FUNCTION_BLOCK AreaOutputEx EXTENDS SectionEx
VAR_IN_OUT
	outputBuffer : ARRAY[*] OF Bundle;
END_VAR
VAR
	passConveyorPos (* AT %I* *) : REAL;
	failConveyorPos (* AT %I* *) : REAL;
	bufferConveyorPos (* AT %I* *) : REAL;
	
	step : (GET_RESULT, CHECK_RESULT, RESET);
	grade : (BYPASS, PASS, FAIL);
END_VAR
VAR
	gradeRequestString : STRING(1000);
	visionTimer : TON;
END_VAR
VAR_STAT CONSTANT
	visionTimeout : TIME := T#10S;
END_VAR

entryRefPos := bufferConveyorPos;
exitRefPos := MAX(passConveyorPos, failConveyorPos);

visionTimer(IN:= , PT:= visionTimeout, Q=> , ET=> );

SUPER^();

METHOD changeRobotsEOAT : BOOL
END_METHOD

METHOD gradeBundle : BOOL
VAR_INPUT
END_VAR
CASE grade OF
	PASS:
		//send to PASS output, LEFT
		
	BYPASS, FAIL:
		//send to FAIL output for manual correction, RIGHT
		
END_CASE
END_METHOD

METHOD initHardware : BOOL
conveyors := ADR(Hardware.allConveyors);
END_METHOD

METHOD PROTECTED load : BOOL
VAR_INPUT
	pair : REFERENCE TO PositionMaterials;
END_VAR
(*
loading takes place while the section is NOT active
materials are loaded for the next incoming bundle, not the current bundle - may differ for each section
*)
END_METHOD

METHOD PROTECTED process : BOOL
VAR
	gradingTcpData : TcpData;
END_VAR
VAR
	visionJson : STRING(1000);
	visionData : VisionFrame;
END_VAR
(*
area output process uses vision PC to determine if a bundle recipe was deployed correctly
1 output for passed bundles, 1 output for failed bundles, center is a buffer queue
*)

CASE step OF
	GET_RESULT:
		setConveyorMode(ConveyorMode.STOP); //stop at camera position (??)
		
		TcpServer1Vision.queue(gradingTcpData);
		step := CHECK_RESULT;
	
	CHECK_RESULT:
		setConveyorMode(ConveyorMode.STOP);
		visionTimer.IN := TRUE;
		
		TcpServer1Vision.fetch(gradingTcpData);
		
		IF NOT BufferIsEmpty(gradingTcpData.binaryData) THEN
			MEMCPY(ADR(visionJson), ADR(gradingTcpData.binaryData), MIN( SIZEOF(visionJson), SIZEOF(gradingTcpData.binaryData) ));
			VisionJsonParser(jsonString:= visionJson, visionData=> visionData);
		END_IF
		
		IF visionTimer.Q THEN
			visionTimer.IN := FALSE;
			grade := BYPASS;
		END_IF
	
	RESET:
		gradeBundle();
		process := TRUE;
		
END_CASE
END_METHOD

METHOD PROTECTED usesProcess : BOOL
VAR
	i : INT;
END_VAR
(*
IF materialsArr = 0 THEN
	RETURN;
END_IF

FOR i:=0 TO GVL.maxPairs BY 1 DO
	IF PositionIsValid(materialsArr[i]) THEN
		usesMaterial := TRUE;
		RETURN;		
	END_IF
END_FOR
*)
END_METHOD

END_FUNCTION_BLOCK

(* stored: Version 1.1.0.1, ProductVersion 3.1.4024.11
   POU AreaOutputEx: Id {50643168-0769-418e-975d-a23807fe5efb}, SpecialFunc None
   Method changeRobotsEOAT: Id {91b2f296-00a1-478b-97a1-d5c66499dfd1}
   Method gradeBundle: Id {6d4cd567-c388-4fb8-ba79-20db376b5be9}
   Method initHardware: Id {1e818c8e-3d72-431c-8cad-784d439be36c}
   Method load: Id {45c420e2-1faa-4c0d-94ba-42357bf20ac7}
   Method process: Id {ae99f37b-a4d0-457e-9e10-86b81ee07c29}
   Method usesProcess: Id {a5c9a7e0-5f20-421f-8c00-954926ed1e8d} *)
